// Mitsubishi GX Works2 project: 西松湘南FLEX   PLC: Q03UDV

PROGRAM FLEXPIWI
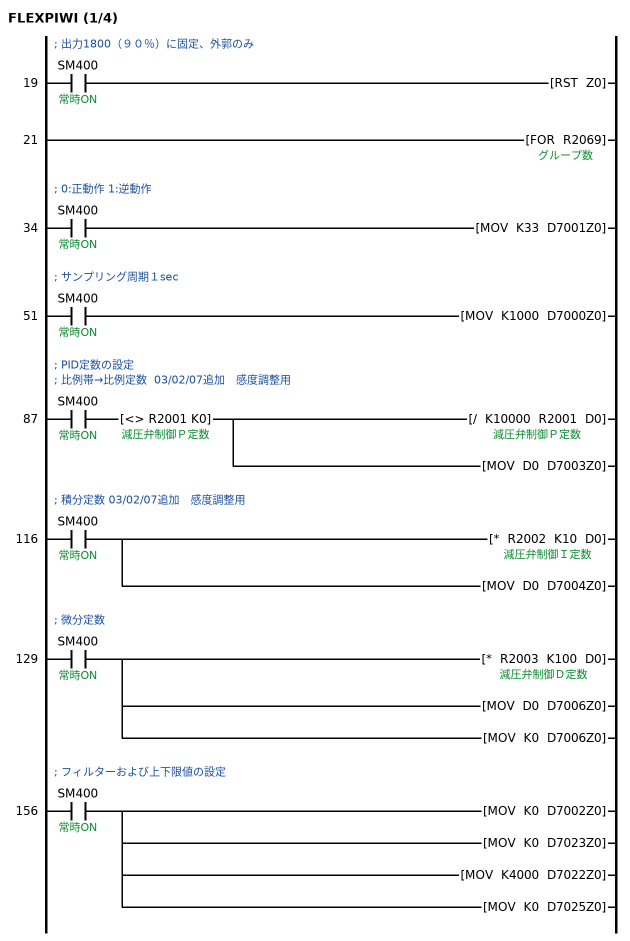
; 出力1800（９０％）に固定、外郭のみ
19    LD      SM400  ; 常時ON
      RST     Z0
21    FOR     R2069  ; グループ数
; 0:正動作 1:逆動作
34    LD      SM400  ; 常時ON
      MOV     K33 D7001Z0
; サンプリング周期１sec
51    LD      SM400  ; 常時ON
      MOV     K1000 D7000Z0
; PID定数の設定
; 比例帯→比例定数  03/02/07追加　感度調整用
87    LD      SM400  ; 常時ON
      AND<>   R2001 K0  ; 減圧弁制御Ｐ定数
      /       K10000 R2001 D0
      MOV     D0 D7003Z0
; 積分定数 03/02/07追加　感度調整用
116   LD      SM400  ; 常時ON
      *       R2002 K10 D0  ; 減圧弁制御Ｉ定数
      MOV     D0 D7004Z0
; 微分定数
129   LD      SM400  ; 常時ON
      *       R2003 K100 D0  ; 減圧弁制御Ｄ定数
      MOV     D0 D7006Z0
      MOV     K0 D7006Z0
; フィルターおよび上下限値の設定
156   LD      SM400  ; 常時ON
      MOV     K0 D7002Z0
      MOV     K0 D7023Z0
      MOV     K4000 D7022Z0
      MOV     K0 D7025Z0
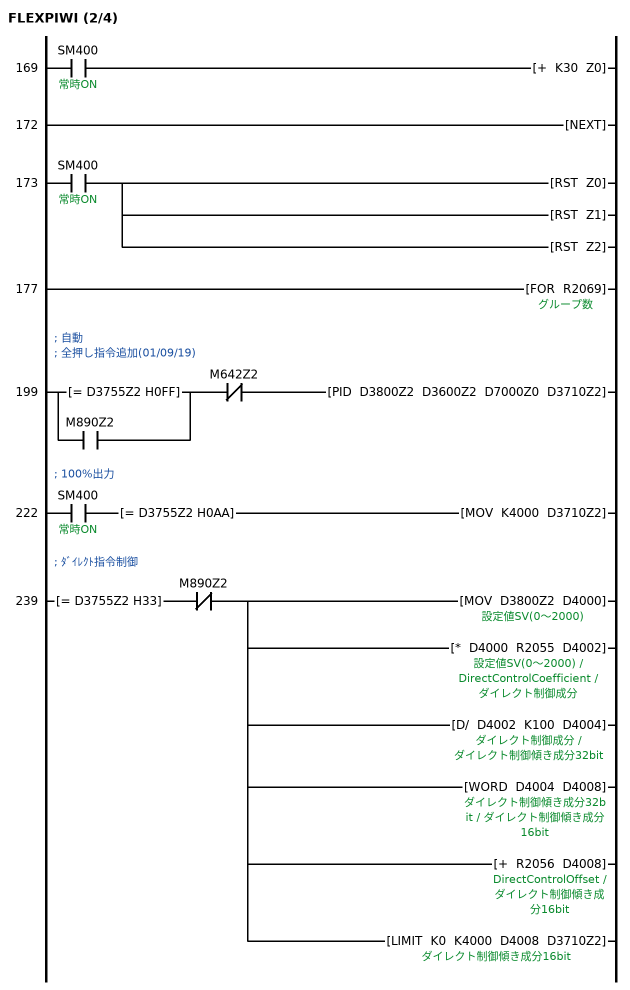
169   LD      SM400  ; 常時ON
      +       K30 Z0
172   NEXT
173   LD      SM400  ; 常時ON
      RST     Z0
      RST     Z1
      RST     Z2
177   FOR     R2069
; 
; 自動
; 全押し指令追加(01/09/19)
199   LD=     D3755Z2 H0FF
      OR      M890Z2
      ANI     M642Z2
      PID     D3800Z2 D3600Z2 D7000Z0 D3710Z2
; 100%出力
222   LD      SM400  ; 常時ON
      AND=    D3755Z2 H0AA
      MOV     K4000 D3710Z2
; ﾀﾞｲﾚｸﾄ指令制御
239   LD=     D3755Z2 H33
      ANI     M890Z2
      MOV     D3800Z2 D4000  ; 設定値SV(0～2000)
      *       D4000 R2055 D4002  ; DirectControlCoefficient / ダイレクト制御成分
      D/      D4002 K100 D4004  ; ダイレクト制御傾き成分32bit
      WORD    D4004 D4008  ; ダイレクト制御傾き成分16bit
      +       R2056 D4008  ; DirectControlOffset
      LIMIT   K0 K4000 D4008 D3710Z2
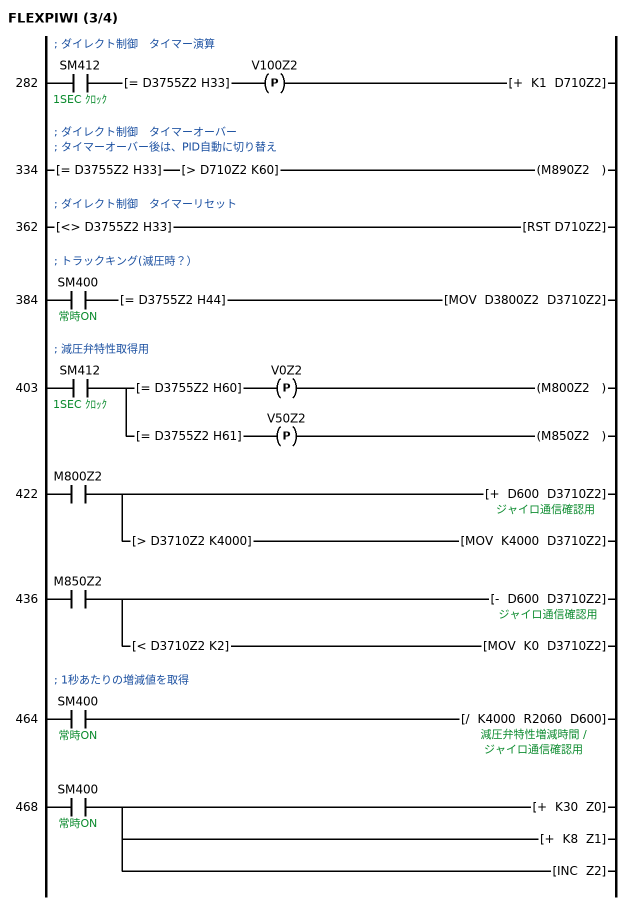
; ダイレクト制御　タイマー演算
282   LD      SM412  ; 1SEC ｸﾛｯｸ
      AND=    D3755Z2 H33
      EGP     V100Z2
      +       K1 D710Z2
; ダイレクト制御　タイマーオーバー
; タイマーオーバー後は、PID自動に切り替え
334   LD=     D3755Z2 H33
      AND>    D710Z2 K60
      OUT     M890Z2
; ダイレクト制御　タイマーリセット
362   LD<>    D3755Z2 H33
      RST     D710Z2
; トラックキング(減圧時？）
384   LD      SM400  ; 常時ON
      AND=    D3755Z2 H44
      MOV     D3800Z2 D3710Z2
; 減圧弁特性取得用
403   LD      SM412  ; 1SEC ｸﾛｯｸ
      MPS
      AND=    D3755Z2 H60
      EGP     V0Z2
      OUT     M800Z2
      MPP
      AND=    D3755Z2 H61
      EGP     V50Z2
      OUT     M850Z2
422   LD      M800Z2
      +       D600 D3710Z2  ; ジャイロ通信確認用
      AND>    D3710Z2 K4000
      MOV     K4000 D3710Z2
436   LD      M850Z2
      -       D600 D3710Z2
      AND<    D3710Z2 K2
      MOV     K0 D3710Z2
; 1秒あたりの増減値を取得
464   LD      SM400  ; 常時ON
      /       K4000 R2060 D600  ; 減圧弁特性増減時間
468   LD      SM400  ; 常時ON
      +       K30 Z0
      +       K8 Z1
      INC     Z2
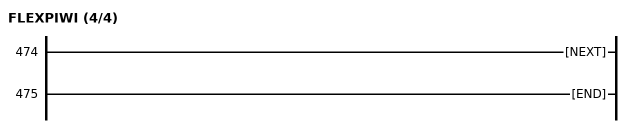
474   NEXT
475   END
END_PROGRAM

PROGRAM FLEXWIN
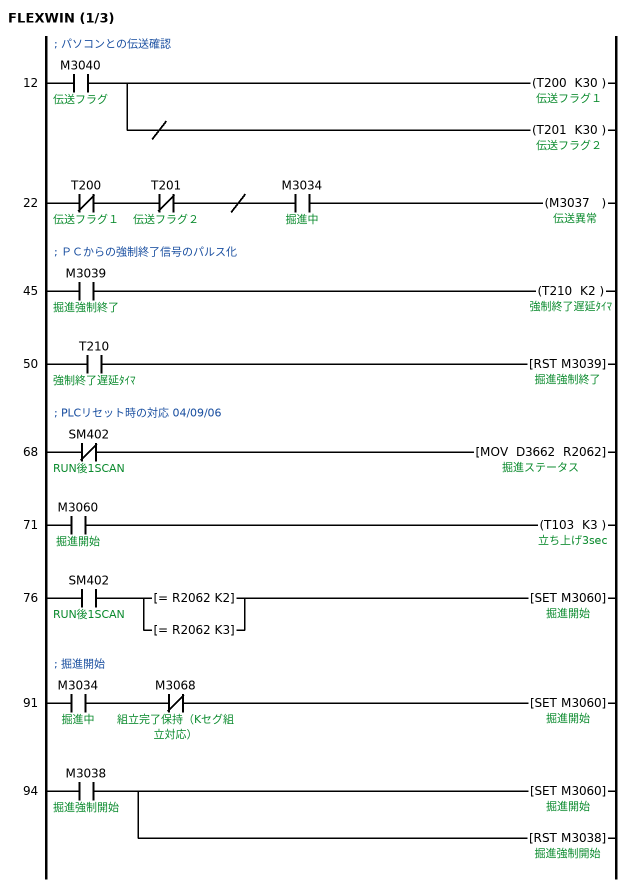
; パソコンとの伝送確認
12    LD      M3040  ; 伝送フラグ
      OUT     T200 K30  ; 伝送フラグ１
      INV
      OUT     T201 K30  ; 伝送フラグ２
22    LDI     T200  ; 伝送フラグ１
      ANI     T201  ; 伝送フラグ２
      INV
      AND     M3034  ; 掘進中
      OUT     M3037  ; 伝送異常
; ＰＣからの強制終了信号のパルス化
45    LD      M3039  ; 掘進強制終了
      OUT     T210 K2  ; 強制終了遅延ﾀｲﾏ
50    LD      T210  ; 強制終了遅延ﾀｲﾏ
      RST     M3039  ; 掘進強制終了
; PLCリセット時の対応 04/09/06
68    LDI     SM402  ; RUN後1SCAN
      MOV     D3662 R2062  ; 掘進ステータス
71    LD      M3060  ; 掘進開始
      OUT     T103 K3  ; 立ち上げ3sec
76    LD      SM402  ; RUN後1SCAN
      LD=     R2062 K2
      OR=     R2062 K3
      ANB
      SET     M3060  ; 掘進開始
; 掘進開始
91    LD      M3034  ; 掘進中
      ANI     M3068  ; 組立完了保持（Kセグ組立対応）
      SET     M3060  ; 掘進開始
94    LD      M3038  ; 掘進強制開始
      SET     M3060  ; 掘進開始
      RST     M3038  ; 掘進強制開始
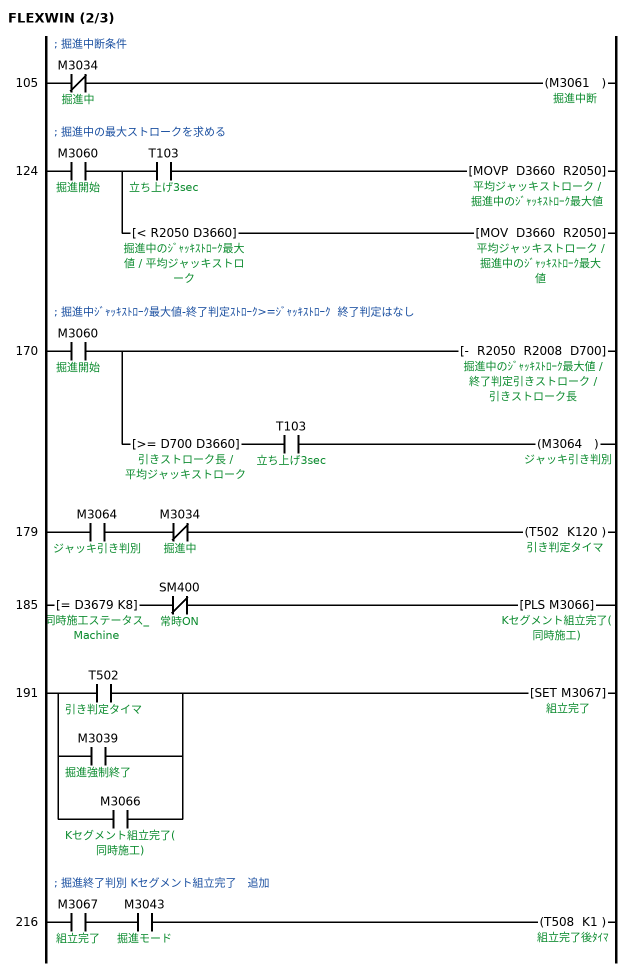
; 掘進中断条件
105   LDI     M3034  ; 掘進中
      OUT     M3061  ; 掘進中断
; 掘進中の最大ストロークを求める
124   LD      M3060  ; 掘進開始
      MPS
      AND     T103  ; 立ち上げ3sec
      MOVP    D3660 R2050  ; 平均ジャッキストローク / 掘進中のｼﾞｬｯｷｽﾄﾛｰｸ最大値
      MPP
      AND<    R2050 D3660  ; 掘進中のｼﾞｬｯｷｽﾄﾛｰｸ最大値 / 平均ジャッキストローク
      MOV     D3660 R2050
; 掘進中ｼﾞｬｯｷｽﾄﾛｰｸ最大値-終了判定ｽﾄﾛｰｸ>=ｼﾞｬｯｷｽﾄﾛｰｸ  終了判定はなし
170   LD      M3060  ; 掘進開始
      -       R2050 R2008 D700  ; 終了判定引きストローク / 引きストローク長
      AND>=   D700 D3660  ; 引きストローク長 / 平均ジャッキストローク
      AND     T103  ; 立ち上げ3sec
      OUT     M3064  ; ジャッキ引き判別
179   LD      M3064  ; ジャッキ引き判別
      ANI     M3034  ; 掘進中
      OUT     T502 K120  ; 引き判定タイマ
185   LD=     D3679 K8  ; 同時施工ステータス_Machine
      ANI     SM400  ; 常時ON
      PLS     M3066  ; Kセグメント組立完了(同時施工)
191   LD      T502  ; 引き判定タイマ
      OR      M3039  ; 掘進強制終了
      OR      M3066  ; Kセグメント組立完了(同時施工)
      SET     M3067  ; 組立完了
; 掘進終了判別 Kセグメント組立完了　追加
216   LD      M3067  ; 組立完了
      AND     M3043  ; 掘進モード
      OUT     T508 K1  ; 組立完了後ﾀｲﾏ
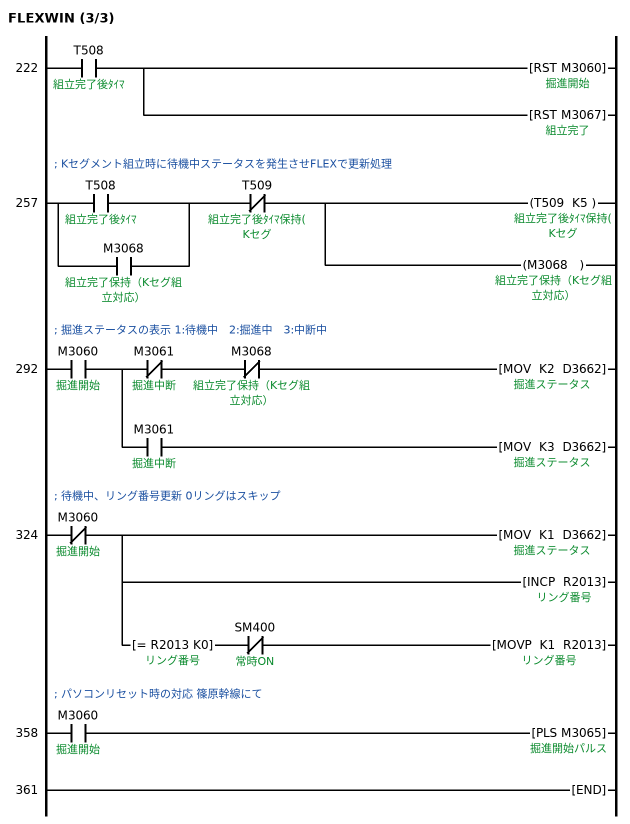
222   LD      T508  ; 組立完了後ﾀｲﾏ
      RST     M3060  ; 掘進開始
      RST     M3067  ; 組立完了
; Kセグメント組立時に待機中ステータスを発生させFLEXで更新処理
257   LD      T508  ; 組立完了後ﾀｲﾏ
      OR      M3068  ; 組立完了保持（Kセグ組立対応）
      ANI     T509  ; 組立完了後ﾀｲﾏ保持(Kセグ
      OUT     T509 K5  ; 組立完了後ﾀｲﾏ保持(Kセグ
      OUT     M3068  ; 組立完了保持（Kセグ組立対応）
; 掘進ステータスの表示 1:待機中　2:掘進中　3:中断中
292   LD      M3060  ; 掘進開始
      MPS
      ANI     M3061  ; 掘進中断
      ANI     M3068  ; 組立完了保持（Kセグ組立対応）
      MOV     K2 D3662
      MPP
      AND     M3061  ; 掘進中断
      MOV     K3 D3662
; 待機中、リング番号更新 0リングはスキップ
324   LDI     M3060  ; 掘進開始
      MOV     K1 D3662
      INCP    R2013  ; リング番号
      AND=    R2013 K0  ; リング番号
      ANI     SM400  ; 常時ON
      MOVP    K1 R2013
; パソコンリセット時の対応 篠原幹線にて
358   LD      M3060  ; 掘進開始
      PLS     M3065  ; 掘進開始パルス
361   END
END_PROGRAM

PROGRAM INOUTWIN
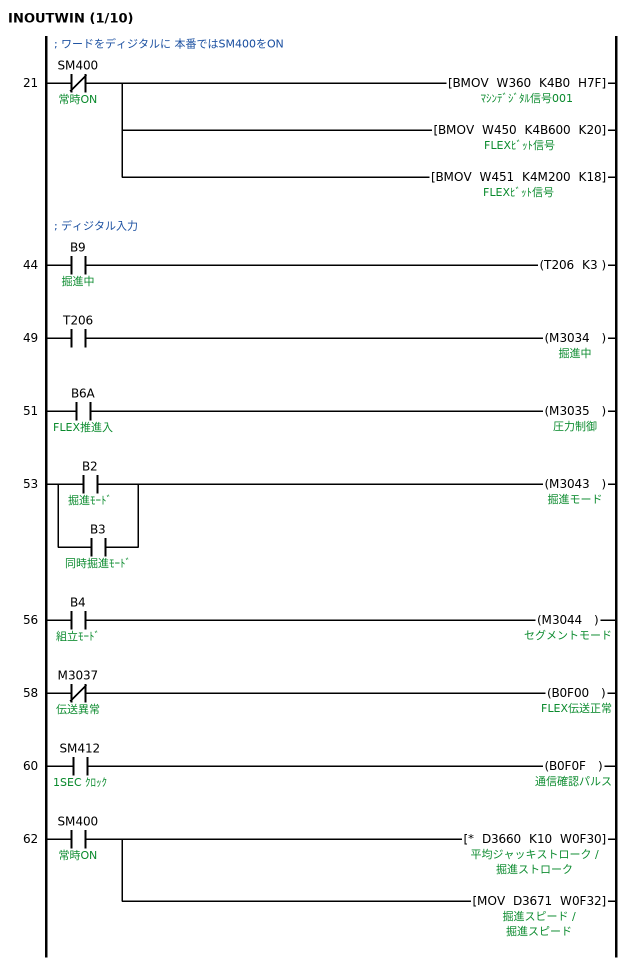
; ワードをディジタルに 本番ではSM400をON
21    LDI     SM400  ; 常時ON
      BMOV    W360 K4B0 H7F  ; ﾏｼﾝﾃﾞｼﾞﾀﾙ信号001 / 中央操作
      BMOV    W450 K4B600 K20  ; FLEXﾋﾞｯﾄ信号 / 通信確認PLS
      BMOV    W451 K4M200 K18  ; FLEXﾋﾞｯﾄ信号 / 中立
; ディジタル入力
44    LD      B9  ; 掘進中
      OUT     T206 K3
49    LD      T206
      OUT     M3034  ; 掘進中
51    LD      B6A  ; FLEX推進入
      OUT     M3035  ; 圧力制御
53    LD      B2  ; 掘進ﾓｰﾄﾞ
      OR      B3  ; 同時掘進ﾓｰﾄﾞ
      OUT     M3043  ; 掘進モード
56    LD      B4  ; 組立ﾓｰﾄﾞ
      OUT     M3044  ; セグメントモード
58    LDI     M3037  ; 伝送異常
      OUT     B0F00  ; FLEX伝送正常
60    LD      SM412  ; 1SEC ｸﾛｯｸ
      OUT     B0F0F  ; 通信確認パルス
62    LD      SM400  ; 常時ON
      *       D3660 K10 W0F30  ; 平均ジャッキストローク / 掘進ストローク
      MOV     D3671 W0F32  ; 掘進スピード / 掘進スピード
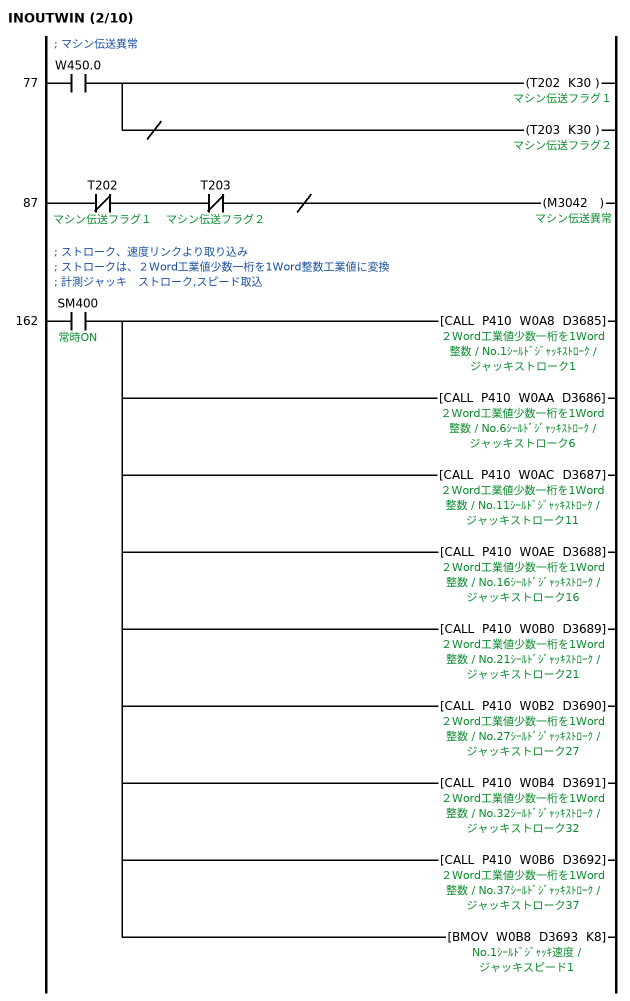
; マシン伝送異常
77    LD      W450.0
      OUT     T202 K30  ; マシン伝送フラグ１
      INV
      OUT     T203 K30  ; マシン伝送フラグ２
87    LDI     T202  ; マシン伝送フラグ１
      ANI     T203  ; マシン伝送フラグ２
      INV
      OUT     M3042  ; マシン伝送異常
; ストローク、速度リンクより取り込み
; ストロークは、２Word工業値少数一桁を1Word整数工業値に変換
; 計測ジャッキ　ストローク,スピード取込
162   LD      SM400  ; 常時ON
      CALL    P410 W0A8 D3685  ; ２Word工業値少数一桁を1Word整数 / No.1ｼｰﾙﾄﾞｼﾞｬｯｷｽﾄﾛｰｸ / ジャッキストローク1
      CALL    P410 W0AA D3686  ; No.6ｼｰﾙﾄﾞｼﾞｬｯｷｽﾄﾛｰｸ / ジャッキストローク6
      CALL    P410 W0AC D3687  ; No.11ｼｰﾙﾄﾞｼﾞｬｯｷｽﾄﾛｰｸ / ジャッキストローク11
      CALL    P410 W0AE D3688  ; No.16ｼｰﾙﾄﾞｼﾞｬｯｷｽﾄﾛｰｸ / ジャッキストローク16
      CALL    P410 W0B0 D3689  ; No.21ｼｰﾙﾄﾞｼﾞｬｯｷｽﾄﾛｰｸ / ジャッキストローク21
      CALL    P410 W0B2 D3690  ; No.27ｼｰﾙﾄﾞｼﾞｬｯｷｽﾄﾛｰｸ / ジャッキストローク27
      CALL    P410 W0B4 D3691  ; No.32ｼｰﾙﾄﾞｼﾞｬｯｷｽﾄﾛｰｸ / ジャッキストローク32
      CALL    P410 W0B6 D3692  ; No.37ｼｰﾙﾄﾞｼﾞｬｯｷｽﾄﾛｰｸ / ジャッキストローク37
      BMOV    W0B8 D3693 K8  ; No.1ｼｰﾙﾄﾞｼﾞｬｯｷ速度 / ジャッキスピード1
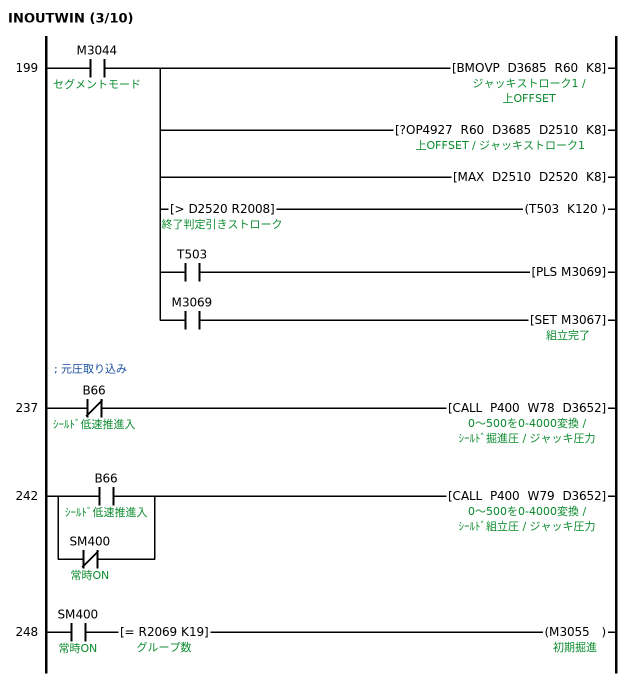
199   LD      M3044  ; セグメントモード
      BMOVP   D3685 R60 K8  ; 上OFFSET
      ?OP4927 R60 D3685 D2510 K8
      MAX     D2510 D2520 K8
      MPS
      AND>    D2520 R2008  ; 終了判定引きストローク
      OUT     T503 K120
      MRD
      AND     T503
      PLS     M3069
      MPP
      AND     M3069
      SET     M3067  ; 組立完了
; 元圧取り込み
237   LDI     B66  ; ｼｰﾙﾄﾞ低速推進入
      CALL    P400 W78 D3652  ; 0～500を0-4000変換 / ｼｰﾙﾄﾞ掘進圧 / ジャッキ圧力
242   LD      B66  ; ｼｰﾙﾄﾞ低速推進入
      ORI     SM400  ; 常時ON
      CALL    P400 W79 D3652  ; ｼｰﾙﾄﾞ組立圧
248   LD      SM400  ; 常時ON
      AND=    R2069 K19  ; グループ数
      OUT     M3055  ; 初期掘進
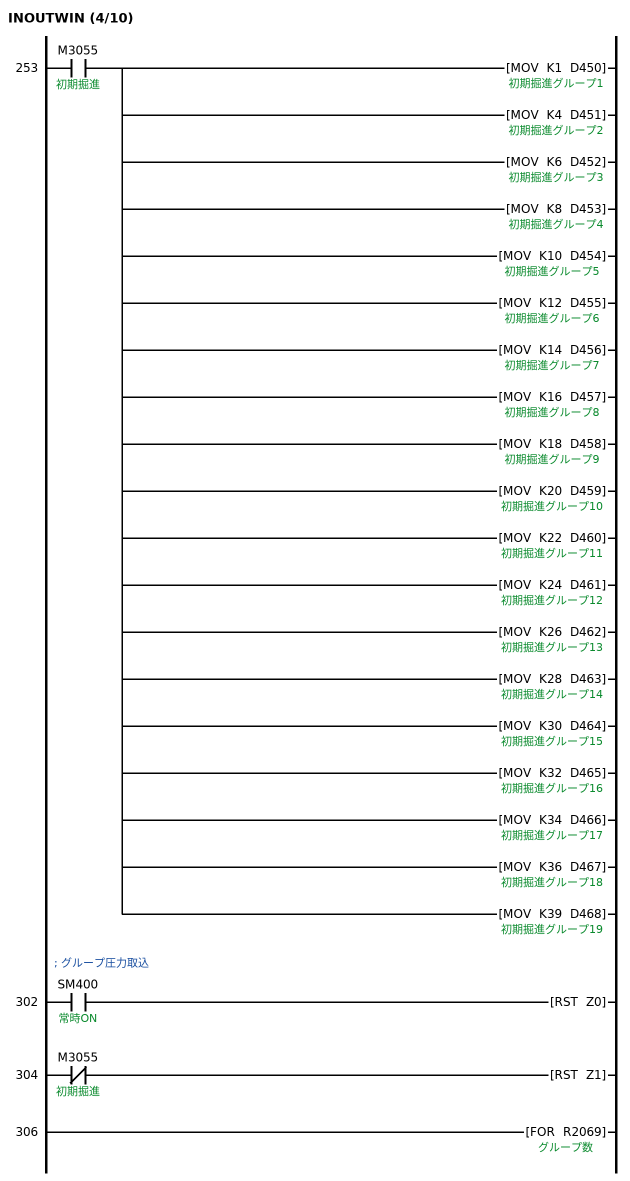
253   LD      M3055  ; 初期掘進
      MOV     K1 D450  ; 初期掘進グループ1
      MOV     K4 D451  ; 初期掘進グループ2
      MOV     K6 D452  ; 初期掘進グループ3
      MOV     K8 D453  ; 初期掘進グループ4
      MOV     K10 D454  ; 初期掘進グループ5
      MOV     K12 D455  ; 初期掘進グループ6
      MOV     K14 D456  ; 初期掘進グループ7
      MOV     K16 D457  ; 初期掘進グループ8
      MOV     K18 D458  ; 初期掘進グループ9
      MOV     K20 D459  ; 初期掘進グループ10
      MOV     K22 D460  ; 初期掘進グループ11
      MOV     K24 D461  ; 初期掘進グループ12
      MOV     K26 D462  ; 初期掘進グループ13
      MOV     K28 D463  ; 初期掘進グループ14
      MOV     K30 D464  ; 初期掘進グループ15
      MOV     K32 D465  ; 初期掘進グループ16
      MOV     K34 D466  ; 初期掘進グループ17
      MOV     K36 D467  ; 初期掘進グループ18
      MOV     K39 D468  ; 初期掘進グループ19
; グループ圧力取込
302   LD      SM400  ; 常時ON
      RST     Z0
304   LDI     M3055  ; 初期掘進
      RST     Z1
306   FOR     R2069
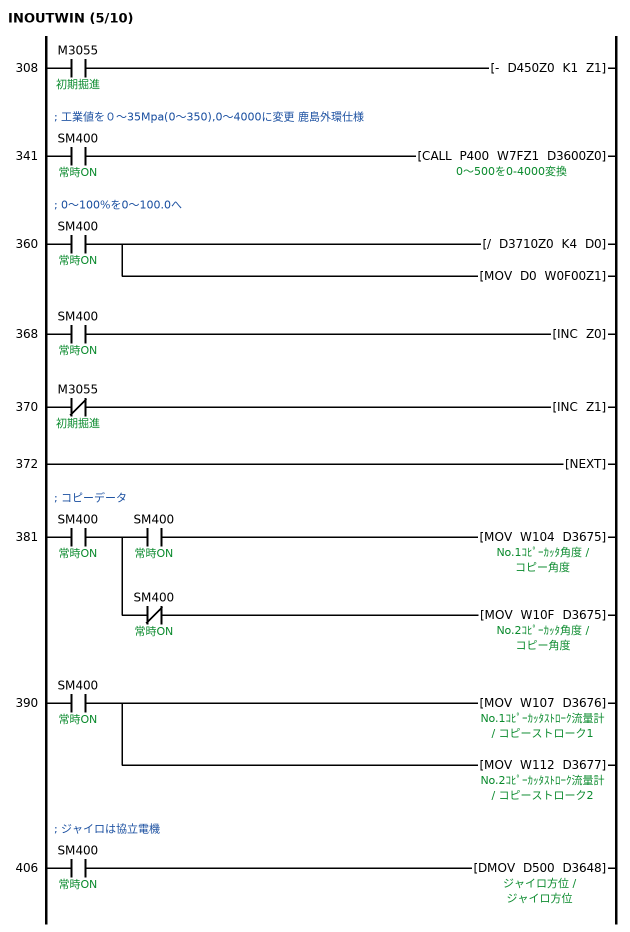
308   LD      M3055  ; 初期掘進
      -       D450Z0 K1 Z1
; 工業値を０～35Mpa(0～350),0～4000に変更 鹿島外環仕様
341   LD      SM400  ; 常時ON
      CALL    P400 W7FZ1 D3600Z0
; 0～100%を0～100.0へ
360   LD      SM400  ; 常時ON
      /       D3710Z0 K4 D0
      MOV     D0 W0F00Z1
368   LD      SM400  ; 常時ON
      INC     Z0
370   LDI     M3055  ; 初期掘進
      INC     Z1
372   NEXT
; コピーデータ
381   LD      SM400  ; 常時ON
      MPS
      AND     SM400  ; 常時ON
      MOV     W104 D3675  ; No.1ｺﾋﾟｰｶｯﾀ角度 / コピー角度
      MPP
      ANI     SM400  ; 常時ON
      MOV     W10F D3675  ; No.2ｺﾋﾟｰｶｯﾀ角度
390   LD      SM400  ; 常時ON
      MOV     W107 D3676  ; No.1ｺﾋﾟｰｶｯﾀｽﾄﾛｰｸ流量計 / コピーストローク1
      MOV     W112 D3677  ; No.2ｺﾋﾟｰｶｯﾀｽﾄﾛｰｸ流量計 / コピーストローク2
; ジャイロは協立電機
406   LD      SM400  ; 常時ON
      DMOV    D500 D3648  ; ジャイロ方位 / ジャイロ方位
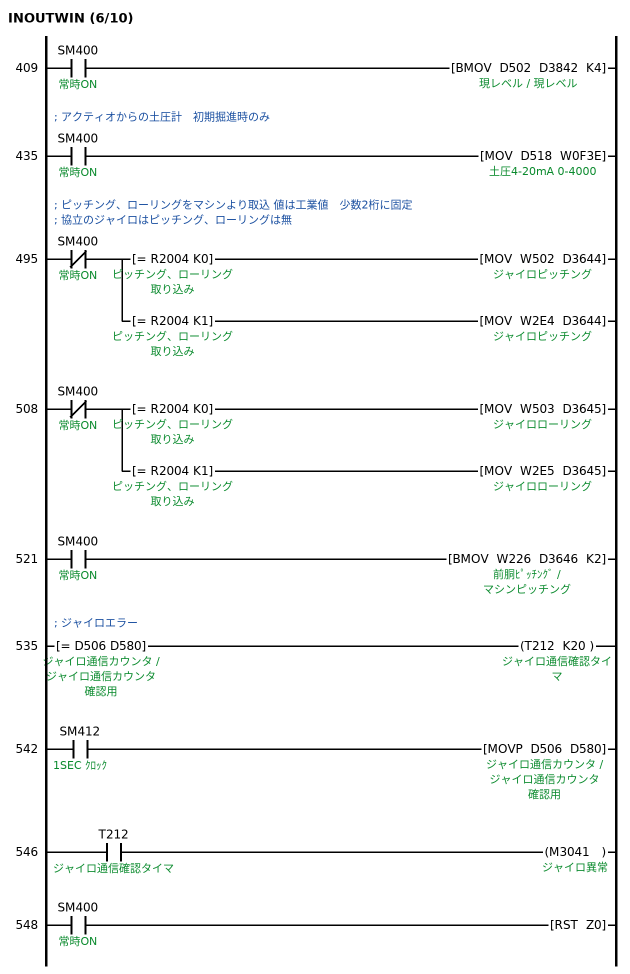
409   LD      SM400  ; 常時ON
      BMOV    D502 D3842 K4  ; 現レベル / 現レベル
; アクティオからの土圧計　初期掘進時のみ
435   LD      SM400  ; 常時ON
      MOV     D518 W0F3E  ; 土圧4-20mA 0-4000
; ピッチング、ローリングをマシンより取込 値は工業値　少数2桁に固定
; 協立のジャイロはピッチング、ローリングは無
495   LDI     SM400  ; 常時ON
      MPS
      AND=    R2004 K0  ; ピッチング、ローリング取り込み
      MOV     W502 D3644  ; ジャイロピッチング
      MPP
      AND=    R2004 K1  ; ピッチング、ローリング取り込み
      MOV     W2E4 D3644
508   LDI     SM400  ; 常時ON
      MPS
      AND=    R2004 K0  ; ピッチング、ローリング取り込み
      MOV     W503 D3645  ; ジャイロローリング
      MPP
      AND=    R2004 K1  ; ピッチング、ローリング取り込み
      MOV     W2E5 D3645
521   LD      SM400  ; 常時ON
      BMOV    W226 D3646 K2  ; 前胴ﾋﾟｯﾁﾝｸﾞ / マシンピッチング
; ジャイロエラー
535   LD=     D506 D580  ; ジャイロ通信カウンタ / ジャイロ通信カウンタ 確認用
      OUT     T212 K20  ; ジャイロ通信確認タイマ
542   LD      SM412  ; 1SEC ｸﾛｯｸ
      MOVP    D506 D580
546   LD      T212  ; ジャイロ通信確認タイマ
      OUT     M3041  ; ジャイロ異常
548   LD      SM400  ; 常時ON
      RST     Z0
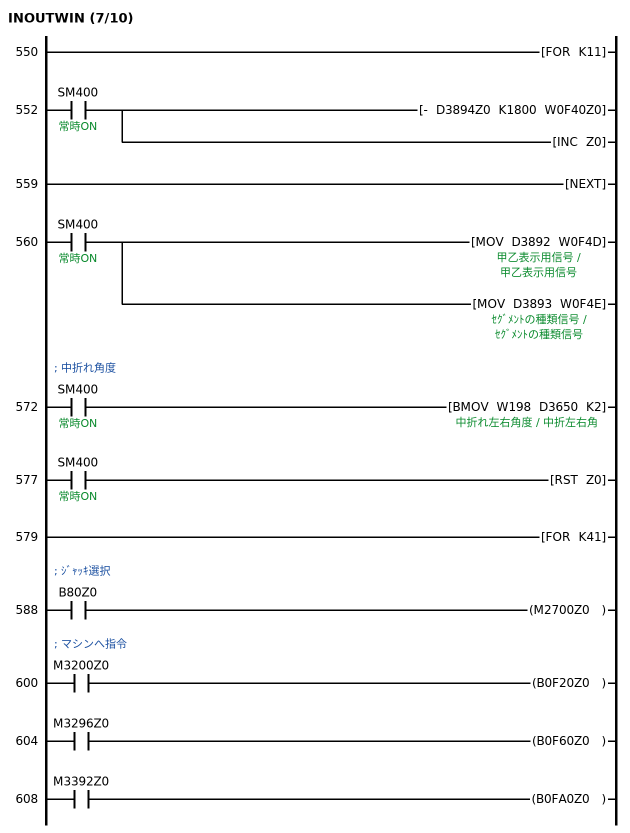
550   FOR     K11
552   LD      SM400  ; 常時ON
      -       D3894Z0 K1800 W0F40Z0
      INC     Z0
559   NEXT
560   LD      SM400  ; 常時ON
      MOV     D3892 W0F4D  ; 甲乙表示用信号 / 甲乙表示用信号
      MOV     D3893 W0F4E  ; ｾｸﾞﾒﾝﾄの種類信号 / ｾｸﾞﾒﾝﾄの種類信号
; 中折れ角度
572   LD      SM400  ; 常時ON
      BMOV    W198 D3650 K2  ; 中折れ左右角度 / 中折左右角
577   LD      SM400  ; 常時ON
      RST     Z0
579   FOR     K41
; ｼﾞｬｯｷ選択
588   LD      B80Z0
      OUT     M2700Z0
; マシンへ指令
600   LD      M3200Z0
      OUT     B0F20Z0
604   LD      M3296Z0
      OUT     B0F60Z0
608   LD      M3392Z0
      OUT     B0FA0Z0
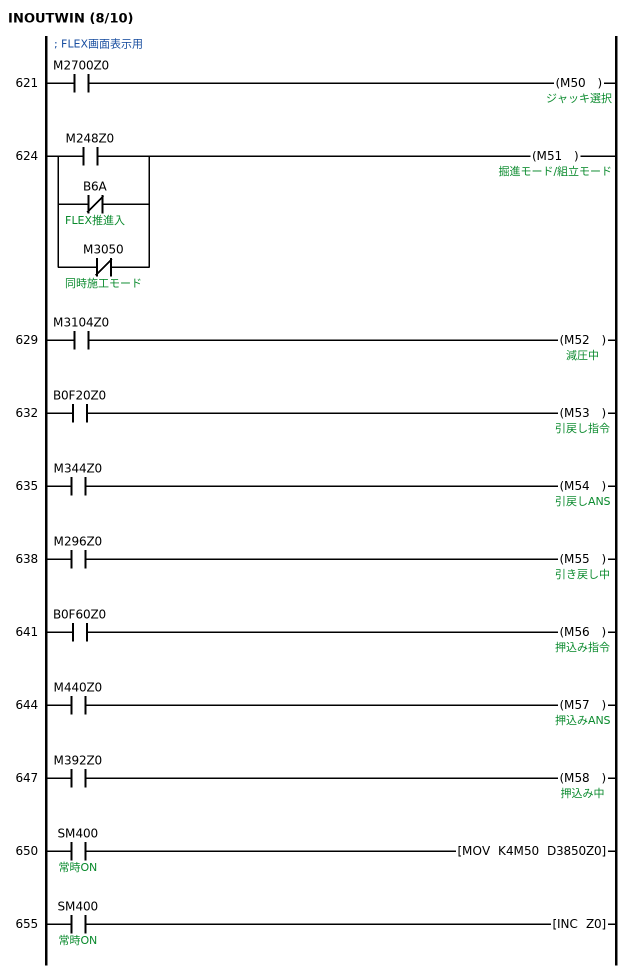
; FLEX画面表示用
621   LD      M2700Z0
      OUT     M50  ; ジャッキ選択
624   LD      M248Z0
      ORI     B6A  ; FLEX推進入
      ORI     M3050  ; 同時施工モード
      OUT     M51  ; 掘進モード/組立モード
629   LD      M3104Z0
      OUT     M52  ; 減圧中
632   LD      B0F20Z0
      OUT     M53  ; 引戻し指令
635   LD      M344Z0
      OUT     M54  ; 引戻しANS
638   LD      M296Z0
      OUT     M55  ; 引き戻し中
641   LD      B0F60Z0
      OUT     M56  ; 押込み指令
644   LD      M440Z0
      OUT     M57  ; 押込みANS
647   LD      M392Z0
      OUT     M58  ; 押込み中
650   LD      SM400  ; 常時ON
      MOV     K4M50 D3850Z0
655   LD      SM400  ; 常時ON
      INC     Z0
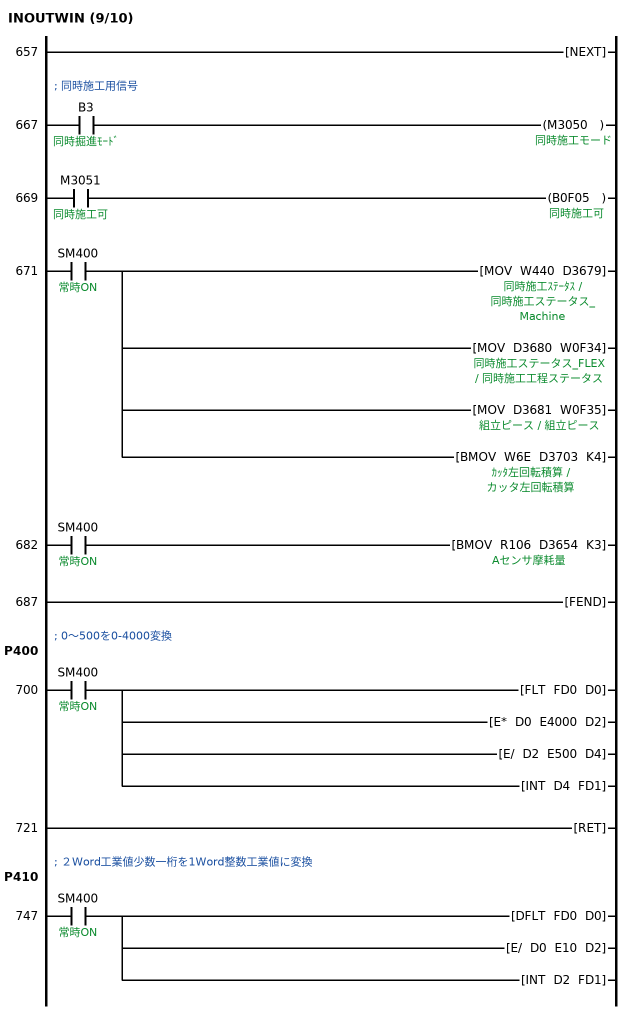
657   NEXT
; 同時施工用信号
667   LD      B3  ; 同時掘進ﾓｰﾄﾞ
      OUT     M3050  ; 同時施工モード
669   LD      M3051  ; 同時施工可
      OUT     B0F05  ; 同時施工可
671   LD      SM400  ; 常時ON
      MOV     W440 D3679  ; 同時施工ｽﾃｰﾀｽ / 同時施工ステータス_Machine
      MOV     D3680 W0F34  ; 同時施工ステータス_FLEX / 同時施工工程ステータス
      MOV     D3681 W0F35  ; 組立ピース / 組立ピース
      BMOV    W6E D3703 K4  ; ｶｯﾀ左回転積算 / カッタ左回転積算
682   LD      SM400  ; 常時ON
      BMOV    R106 D3654 K3  ; Aセンサ摩耗量
687   FEND
      P400
; 0～500を0-4000変換
700   LD      SM400  ; 常時ON
      FLT     FD0 D0
        [note] スケール上限
      E*      D0 E4000 D2
      E/      D2 E500 D4
      INT     D4 FD1
721   RET
      P410
; ２Word工業値少数一桁を1Word整数工業値に変換
747   LD      SM400  ; 常時ON
      DFLT    FD0 D0
        [note] スケール上限
      E/      D0 E10 D2
      INT     D2 FD1
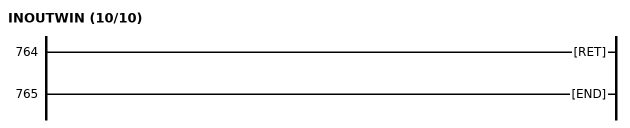
764   RET
765   END
END_PROGRAM

PROGRAM SIMLAT
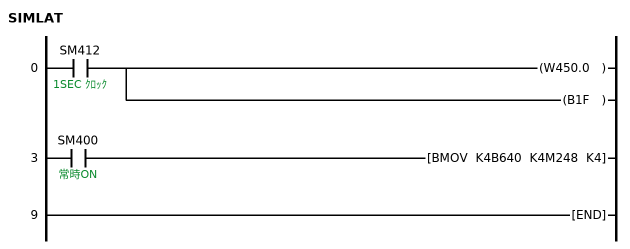
0     LD      SM412  ; 1SEC ｸﾛｯｸ
      OUT     W450.0
      OUT     B1F
3     LD      SM400  ; 常時ON
      BMOV    K4B640 K4M248 K4  ; No.1ｼｰﾙﾄﾞｼﾞｬｯｷ掘進中
9     END
END_PROGRAM

PROGRAM GYRO
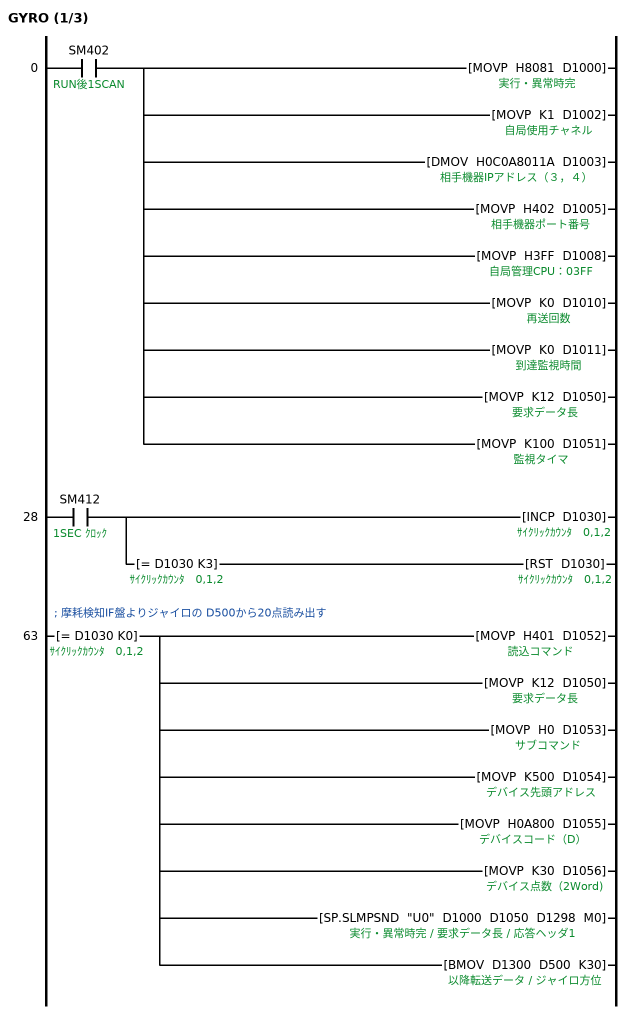
0     LD      SM402  ; RUN後1SCAN
      MOVP    H8081 D1000  ; 実行・異常時完
      MOVP    K1 D1002  ; 自局使用チャネル
      DMOV    H0C0A8011A D1003  ; 相手機器IPアドレス（３，４）
      MOVP    H402 D1005  ; 相手機器ポート番号
      MOVP    H3FF D1008  ; 自局管理CPU：03FF
      MOVP    K0 D1010  ; 再送回数
      MOVP    K0 D1011  ; 到達監視時間
      MOVP    K12 D1050  ; 要求データ長
      MOVP    K100 D1051  ; 監視タイマ
28    LD      SM412  ; 1SEC ｸﾛｯｸ
      INCP    D1030  ; ｻｲｸﾘｯｸｶｳﾝﾀ　0,1,2
      AND=    D1030 K3  ; ｻｲｸﾘｯｸｶｳﾝﾀ　0,1,2
      RST     D1030  ; ｻｲｸﾘｯｸｶｳﾝﾀ　0,1,2
; 摩耗検知IF盤よりジャイロの D500から20点読み出す
63    LD=     D1030 K0  ; ｻｲｸﾘｯｸｶｳﾝﾀ　0,1,2
      MOVP    H401 D1052  ; 読込コマンド
        [note] 読みしコマンド
      MOVP    K12 D1050
      MOVP    H0 D1053  ; サブコマンド
      MOVP    K500 D1054  ; デバイス先頭アドレス
      MOVP    H0A800 D1055  ; デバイスコード（D）
      MOVP    K30 D1056  ; デバイス点数（2Word)
      SP.SLMPSND "U0" D1000 D1050 D1298 M0  ; 応答ヘッダ1
      BMOV    D1300 D500 K30  ; 以降転送データ / ジャイロ方位
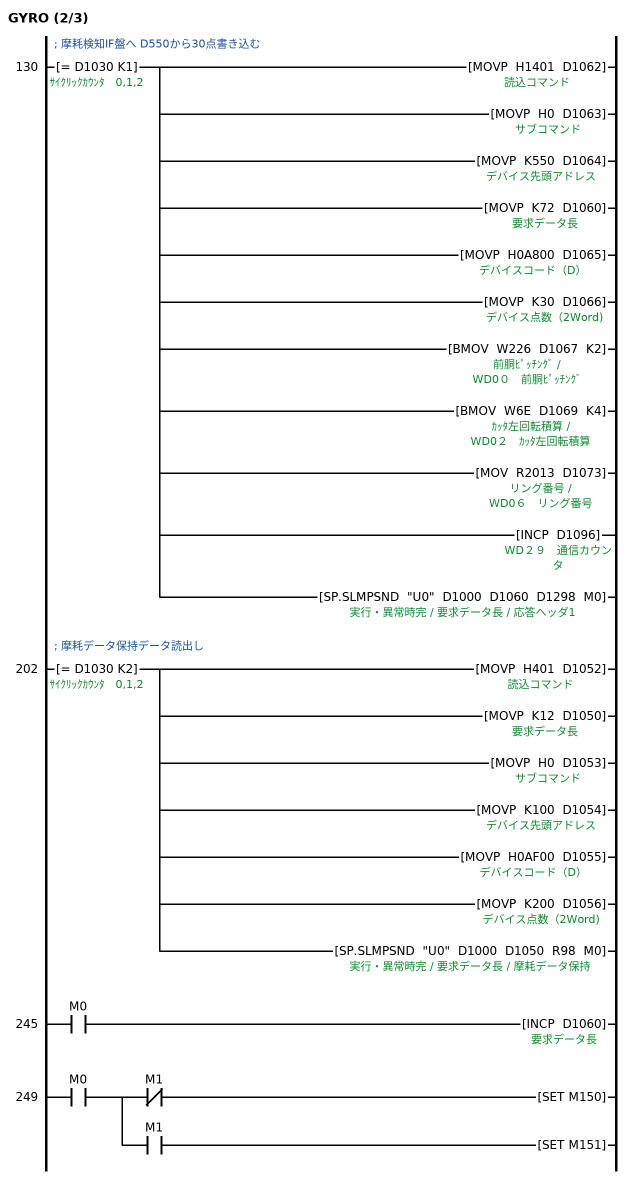
; 摩耗検知IF盤へ D550から30点書き込む
130   LD=     D1030 K1  ; ｻｲｸﾘｯｸｶｳﾝﾀ　0,1,2
      MOVP    H1401 D1062  ; 読込コマンド
        [note] 書き込みコマンド
      MOVP    H0 D1063  ; サブコマンド
      MOVP    K550 D1064  ; デバイス先頭アドレス
      MOVP    K72 D1060  ; 要求データ長
      MOVP    H0A800 D1065  ; デバイスコード（D）
      MOVP    K30 D1066  ; デバイス点数（2Word)
      BMOV    W226 D1067 K2  ; 前胴ﾋﾟｯﾁﾝｸﾞ / WD0０　前胴ﾋﾟｯﾁﾝｸﾞ
      BMOV    W6E D1069 K4  ; ｶｯﾀ左回転積算 / WD0２　ｶｯﾀ左回転積算
      MOV     R2013 D1073  ; リング番号 / WD0６　リング番号
      INCP    D1096  ; WD２９　通信カウンタ
      SP.SLMPSND "U0" D1000 D1060 D1298 M0
; 摩耗データ保持データ読出し
202   LD=     D1030 K2  ; ｻｲｸﾘｯｸｶｳﾝﾀ　0,1,2
      MOVP    H401 D1052
        [note] 読みしコマンド
      MOVP    K12 D1050
      MOVP    H0 D1053
      MOVP    K100 D1054
      MOVP    H0AF00 D1055
      MOVP    K200 D1056
      SP.SLMPSND "U0" D1000 D1050 R98 M0  ; 摩耗データ保持
245   LD      M0
      INCP    D1060
249   LD      M0
      MPS
      ANI     M1
      SET     M150
      MPP
      AND     M1
      SET     M151
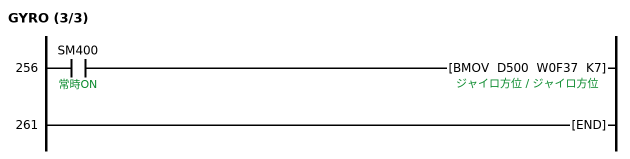
256   LD      SM400  ; 常時ON
      BMOV    D500 W0F37 K7  ; ジャイロ方位
261   END
END_PROGRAM

PROGRAM MCPRTCL
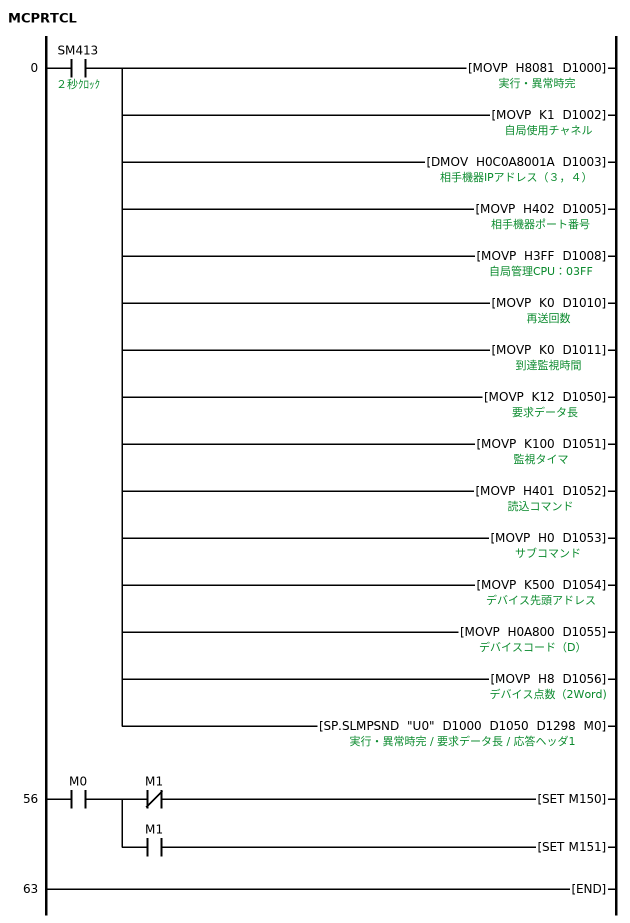
0     LD      SM413  ; ２秒ｸﾛｯｸ
      MOVP    H8081 D1000  ; 実行・異常時完
      MOVP    K1 D1002  ; 自局使用チャネル
      DMOV    H0C0A8001A D1003  ; 相手機器IPアドレス（３，４）
      MOVP    H402 D1005  ; 相手機器ポート番号
      MOVP    H3FF D1008  ; 自局管理CPU：03FF
      MOVP    K0 D1010  ; 再送回数
      MOVP    K0 D1011  ; 到達監視時間
      MOVP    K12 D1050  ; 要求データ長
      MOVP    K100 D1051  ; 監視タイマ
      MOVP    H401 D1052  ; 読込コマンド
      MOVP    H0 D1053  ; サブコマンド
      MOVP    K500 D1054  ; デバイス先頭アドレス
      MOVP    H0A800 D1055  ; デバイスコード（D）
      MOVP    H8 D1056  ; デバイス点数（2Word)
      SP.SLMPSND "U0" D1000 D1050 D1298 M0  ; 応答ヘッダ1
56    LD      M0
      MPS
      ANI     M1
      SET     M150
      MPP
      AND     M1
      SET     M151
63    END
END_PROGRAM

// device comments not shown above
D710  ; グループ1ダイレクト時間
D3710  ; グループ1圧力MV
D3894  ; 1ピース目標角度
W0F40  ; 1ピース目標角度
